PROGRAM drives
VAR
	//Small Drive
	aSmallDrive					: AXIS_REF; //initilization of asmallDrive axis
	MC_Power_aSmallDrive		: MC_Power; // linking to the FB
	MC_JOG_aSmallDrive			: MC_Jog;   //linking to the FB
	
	//LargeDrive
	alargeDrive					: AXIS_REF;	
	MC_Power_aLargeDrive		: MC_Power;
	MC_JOG_aLargeDrive			: MC_Jog;
	
	Read_Actual_position		: MC_ReadActualPosition;
	ActualPositionArray 				: ARRAY [1..1000000] OF REAL;
	Reset_largeDrive			: MC_Reset;
	Reset_smallDrive			: MC_Reset;
	
	Index 						: INT:=1;
	Position					: REAL;

	
	
	TIMER: TON;
	FILEWRITE: FB_FileWrite;
END_VAR

//conditional statement for switching the RGB, Red for Emergency Stop , Green for motor 1 and Orange for motor2
IF NOT cabinet.emergencysw THEN
	Reset_largeDrive.Execute 			:= FALSE;
	Reset_smallDrive.Execute			:= FALSE;
    cabinet.redlight    				:= TRUE;
    cabinet.greenlight  				:= FALSE;
    cabinet.orangelight 				:= FALSE;
ELSIF cabinet.emergencysw AND cabinet.selector1 THEN
	Reset_smallDrive.Execute			:= TRUE;
    cabinet.redlight    				:= FALSE;
    cabinet.greenlight  				:= TRUE;
    cabinet.orangelight 				:= FALSE;   
ELSIF cabinet.emergencysw AND cabinet.selector2 THEN 
	Reset_largeDrive.Execute			:= TRUE;
    cabinet.redlight   					:= FALSE;
    cabinet.greenlight  				:= FALSE;
    cabinet.orangelight 				:= TRUE; 
END_IF

//Emergency switch to stop the motors
IF cabinet.emergencysw THEN
    drives.MC_Power_aSmallDrive.Enable := TRUE;
	drives.MC_Power_aLargeDrive.Enable := TRUE;
ELSE	
	drives.MC_Power_aSmallDrive.Enable := FALSE;
	drives.MC_Power_aLargeDrive.Enable := FALSE;
END_IF


//Selector conditonal statement
IF cabinet.selector1 THEN
	
	driveController.smallDrive.xForward := cabinet.motor1fwd;
	driveController.smallDrive.xReverse := cabinet.motor1rev;
ELSE
	driveController.largeDrive.xForward := cabinet.motor2fwd;
	driveController.largeDrive.xReverse := cabinet.motor2rev;	
END_IF

//FB to read the positon of the large servo motor
Read_Actual_position(
	Axis								:= alargeDrive, 
	Enable								:= TRUE , 
	Valid=> , 
	Busy=> , 
	Error=> , 
	ErrorID=> , 
	Position							 => driveController.largeDrive.actualposition);
	
	
	
//Fb to reset the large servo motor
Reset_largeDrive(
	Axis								:= alargeDrive, 
	Execute								:=  , 
	Done=> , 
	Busy=> , 
	Error=> , 
	ErrorID=> );

//FB to reset the small servo motor
Reset_smallDrive(
	Axis								:=aSmallDrive , 
	Execute								:= , 
	Done=> , 
	Busy=> , 
	Error=> , 
	ErrorID=> );


//small motor power and jog
MC_Power_aSmallDrive(
		Axis							:= aSmallDrive, 
		Enable							:= , 
		Enable_Positive					:= TRUE, 
		Enable_Negative					:= TRUE, 
		Override						:= 100, 
		BufferMode						:= , 
		Options							:= , 
		Status							=> , 
		Busy							=> , 
		Active							=> , 
		Error							=> , 
		ErrorID							=> );
	
MC_JOG_aSmallDrive(
		Axis							:= aSmallDrive, 
		JogForward						:= driveController.smallDrive.xForward, 
		JogBackwards					:= driveController.smallDrive.xReverse, 
		Mode							:= E_JogMode.MC_JOGMODE_CONTINOUS,
		//Position:= , 
		Velocity						:= 500, 
		Acceleration					:= 15000, 
		Deceleration					:= 15000, 
		Jerk							:= 15000, 
		Done							=> , 
		Busy							=> , 
		Active							=> , 
		CommandAborted					=> , 
		Error							=> , 
		ErrorID							=> );
	


//large drive Power and jog
MC_Power_aLargeDrive(
		Axis							:=alargeDrive , 
		Enable							:= , 
		Enable_Positive					:=TRUE , 
		Enable_Negative					:=TRUE , 
		Override						:=100 , 
		BufferMode						:= , 
		Options							:= , 
		Status							=> , 
		Busy							=> , 
		Active							=> , 
		Error							=> , 
		ErrorID							=> );
		
	MC_JOG_aLargeDrive(
		Axis							:= alargeDrive, 
		JogForward						:= driveController.largeDrive.xForward, 
		JogBackwards					:= driveController.largeDrive.xReverse, 
		Mode							:= E_JogMode.MC_JOGMODE_CONTINOUS,
		//Position:= , 
		Velocity						:= 100, 
		Acceleration					:= 1000, 
		Deceleration					:= 1000, 
		Jerk							:= 1000, 
		Done							=> , 
		Busy							=> , 
		Active							=> , 
		CommandAborted					=> , 
		Error							=> , 
		ErrorID							=> );

TIMER(IN:= , PT:= T#5S , Q=> , ET=>  );		
IF driveController.largeDrive.xForward OR driveController.largeDrive.xReverse THEN
	TIMER(IN := TRUE);
END_IF

IF TIMER.Q THEN
    Position := driveController.largeDrive.actualposition;
    ActualPositionArray[Index] := Position;
    Index := Index + 1;
	Timer(IN := FALSE);
	
	
	IF Index > 100000 THEN
        Timer(IN := FALSE);  (* Stop the timer when 100 values are stored *)
    END_IF
	
END_IF

FILEWRITE(
	sNetId:= , 
	hFile:= , 
	pWriteBuff:= , 
	cbWriteLen:= , 
	bExecute:= , 
	tTimeout:= , 
	bBusy=> , 
	bError=> , 
	nErrId=> , 
	cbWrite=> );

END_PROGRAM

(* stored: Version 1.1.0.1, ProductVersion 3.1.4024.12
   POU drives: Id {dede6169-9d00-441b-82ba-083c9992ede6}, SpecialFunc None *)
